# EPICS substitutions: db/ecat2ek1101.substitutions
file ecat2ekxxxxID.template
{
	pattern {NULL}
		{NULL}

}

file ecat2slave.template
{
	pattern {DTYP}
		{EK1101}
}
